TYPE "Positioning_DOL_Machine_CIn"
VERSION : 0.1
// Block: Positioning_DOL_Machine_CIn
   STRUCT
      Manager : Positioning_DOL_Machine_Manager;
      MinusExtEnable : Bool;
      PlusExtEnable : Bool;
      ExternalPowerOn : Bool;
      ExternalAlarms : Bool;
      PositionLimits : Struct
         EnableMin : Bool;
         PosMin : LReal;
         EnableMax : Bool;
         PosMax : LReal;
      END_STRUCT;
   END_STRUCT;

END_TYPE
